Fanuc KAREL source: kd00064.KL

PROGRAM KD00064
%STACKSIZE=65535
%PRIORITY=65535
%NOLOCKGROUP
VAR
I : INTEGER
J : INTEGER
B : BOOLEAN
R : REAL
S : STRING[80]
BEGIN
-- UNRESOLVED_PC line 10 opcodes [9D 81 18 9D 1B 9D 12 9C 13 04] marker_code=0
END KD00064
